TYPE ST_P_SAVE_MESDAT :
STRUCT
	SetIndex:				BOOL;
	Index:					INT;
	Barcode:				INT;
END_STRUCT
END_TYPE

(* stored: Version 1.1.0.1, ProductVersion 3.1.4024.10
   DUT ST_P_SAVE_MESDAT: Id {215f6cfd-c38b-43f9-bcfa-a1ab3077864b} *)
